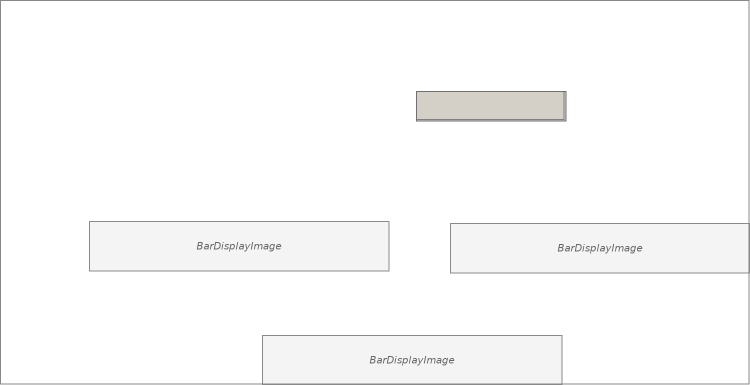
VISUALIZATION Visualization  // 750x385
    BarDisplayImage (89,221 300x50), value: MAIN.fbSlicer.AxisM1.NcToPlc.ActPos, style: BarDisplayImage-Gray, scale format: %.1f, scale 0..100
    BarDisplayImage (450,223 300x50), value: MAIN.fbSlicer.AxisM1s.NcToPlc.ActPos, style: BarDisplayImage-Gray, scale format: %.1f, scale 0..100
    BarDisplayImage (262,335 300x50), value: MAIN.fbSlicer.AxisM2.NcToPlc.ActPos, style: BarDisplayImage-Gray, scale format: %.1f, scale 0..100
    Button (416,91 150x30)
        tap MAIN.bStartButton
END_VISUALIZATION

(* stored: Version 1.1.0.1, ProductVersion 3.1.4024.12
   Visu Visualization: Id {bd51f1f8-8971-4e21-a1f3-e28f6d6dbd75} *)
